// TIA Portal V20 export
DATA_BLOCK "DB_Digital_Inputs"   // DB1
{ S7_Optimized_Access := 'TRUE' }
// stored: MemoryReserve 100
   VAR
      Digital_Input_0 : Bool;
      Digital_Input_1 : Bool;
      Digital_Input_2 : Bool;
      Digital_Input_3 : Bool;
      Digital_Input_4 : Bool;
      Digital_Input_5 : Bool;
      Digital_Input_6 : Bool;
      Digital_Input_7 : Bool;
      Digital_Input_8 : Bool;
      Digital_Input_9 : Bool;
      Digital_Input_10 : Bool;
      Digital_Input_11 : Bool;
      Digital_Input_12 : Bool;
      Digital_Input_13 : Bool;
   END_VAR
BEGIN
END_DATA_BLOCK
